SYSTEM TEST_ARRAY_IO (* Test ARRAY_IN,ARRAY_OUT *)
  (* Standard: 61499-2 *)
  (* Version 0.0, 2000-05-27, JHC, Rockwell Automation *)
  DEVICE ARRAY_IO : FRAME_DEVICE
    RESOURCE RES1 : PANEL_RESOURCE
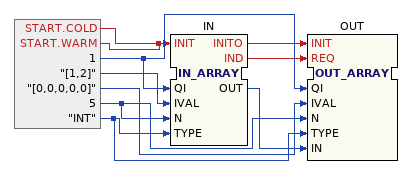
      FBS
        IN : IN_ARRAY;
        OUT : OUT_ARRAY;
      END_FBS
      EVENT_CONNECTIONS
        START.COLD TO IN.INIT;
        START.WARM TO IN.INIT;
        IN.INITO TO OUT.INIT;
        IN.IND TO OUT.REQ;
      END_CONNECTIONS
      DATA_CONNECTIONS
        1 TO IN.QI;
        1 TO OUT.QI;
        "[1,2]" TO IN.IVAL;
        "[0,0,0,0,0]" TO OUT.IVAL;
        5 TO IN.N;
        5 TO OUT.N;
        "INT" TO IN.TYPE;
        "INT" TO OUT.TYPE;
        IN.OUT TO OUT.IN;
      END_CONNECTIONS
    END_RESOURCE
  END_DEVICE
  DATA_CONNECTIONS (* parameter values *)
    [100,100,200,100] TO ARRAY_IO.BOUNDS;
    [1,1] TO ARRAY_IO.GRID;
  END_CONNECTIONS
END_SYSTEM
